FUNCTION_BLOCK IX
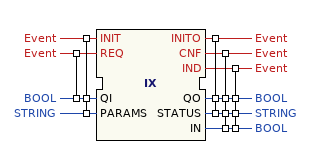
  EVENT_INPUT
    INIT WITH QI, PARAMS;
    REQ WITH QI;
  END_EVENT
  EVENT_OUTPUT
    INITO WITH QO, STATUS;
    CNF WITH QO, STATUS, IN;
    IND WITH QO, STATUS, IN;
  END_EVENT
  VAR_INPUT
    QI : BOOL;
    PARAMS : STRING;
  END_VAR
  VAR_OUTPUT
    QO : BOOL;
    STATUS : STRING;
    IN : BOOL;
  END_VAR
END_FUNCTION_BLOCK
